# B&R Automation Studio project TD52 (part 59)

#### AC_SS.c
```c
/********************************************************************
 * COPYRIGHT -- Bernecker + Rainer Industrie-Elektronik Ges.m.b.H.
 ********************************************************************
 * Program: AC_SS
 * File: AC_SS.c
 * Author: 105055527
 * Created: Thu May 19 13:50:06 2016
 ********************************************************************
 * Implementation of program AC_SS
 ********************************************************************
 * Generated with B&R Automation Studio Target for Simulink V5.0
 * (ERT based)
 ********************************************************************/
#include "AC_SS.h"
#include "AC_SS_private.h"

/*  Defines */

/*  Data Types */

/**************************** GLOBAL DATA *************************************/
/*  Definitions */

/*  Declarations  */

/***************************** FILE SCOPE DATA ********************************/

/*************************** FUNCTIONS ****************************************/

/*
 * Initial conditions for atomic system:
 *    '<S13>/Filter'
 *    '<S19>/Filter'
 *    '<S25>/Filter'
 *    '<S31>/Filter'
 *    '<S37>/Filter'
 *    '<S43>/Filter'
 *    '<S49>/Filter'
 *    '<S55>/Filter'
 */
void AC_SS_Filter_Init(real32_T rtu_x0, rtDW_Filter_AC_SS *localDW, struct SS* inst)
{
  /* InitializeConditions for DiscreteIntegrator: '<S14>/Discrete-Time Integrator' */
  localDW->DiscreteTimeIntegrator_DSTATE = rtu_x0;
}

/*
 * Output and update for atomic system:
 *    '<S13>/Filter'
 *    '<S19>/Filter'
 *    '<S25>/Filter'
 *    '<S31>/Filter'
 *    '<S37>/Filter'
 *    '<S43>/Filter'
 *    '<S49>/Filter'
 *    '<S55>/Filter'
 */
void AC_SS_Filter(real32_T rtu_in, real32_T rtu_T_filt, boolean_T rtu_reset,
                  real32_T rtu_x0, rtB_Filter_AC_SS *localB, rtDW_Filter_AC_SS
                  *localDW, struct SS* inst)
{
  /* local block i/o variables */
  real32_T rtb_Divide4;
  real32_T tmp;

  /* Switch: '<S15>/Switch' incorporates:
   *  Abs: '<S15>/Abs'
   *  RelationalOperator: '<S15>/Relational Operator'
   */
  if (2.22044605E-16F >= (real32_T)fabs(rtu_T_filt)) {
    tmp = 2.22044605E-16F;
  } else {
    tmp = rtu_T_filt;
  }

  /* End of Switch: '<S15>/Switch' */

  /* Product: '<S14>/Divide4' incorporates:
   *  Sum: '<S14>/Sum4'
   */
  rtb_Divide4 = (rtu_in - localDW->DiscreteTimeIntegrator_DSTATE) / tmp;

  /* DiscreteIntegrator: '<S14>/Discrete-Time Integrator' */
  if (rtu_reset || (localDW->DiscreteTimeIntegrator_PrevRese != 0)) {
    localDW->DiscreteTimeIntegrator_DSTATE = rtu_x0;
  }

  localB->DiscreteTimeIntegrator = 0.005F * rtb_Divide4 +
    localDW->DiscreteTimeIntegrator_DSTATE;

  /* End of DiscreteIntegrator: '<S14>/Discrete-Time Integrator' */

  /* Update for DiscreteIntegrator: '<S14>/Discrete-Time Integrator' */
  if (!rtu_reset) {
    localDW->DiscreteTimeIntegrator_DSTATE = 0.005F * rtb_Divide4 +
      localB->DiscreteTimeIntegrator;
  }

  if (rtu_reset) {
    localDW->DiscreteTimeIntegrator_PrevRese = 1;
  } else {
    localDW->DiscreteTimeIntegrator_PrevRese = 0;
  }

  /* End of Update for DiscreteIntegrator: '<S14>/Discrete-Time Integrator' */
}

/* Model step function */
void AC_SS_step(struct BlockIO_AC_SS *AC_SS_B, struct D_Work_AC_SS *AC_SS_DWork,
                ExternalOutputs_AC_SS *AC_SS_Y, struct SS* inst)
{
  /* local block i/o variables */
  real32_T rtb_rAct;
  real32_T rtb_rTi_Filt;
  real32_T rtb_rAct_h;
  real32_T rtb_rTi_Filt_h;
  real32_T rtb_rAct_hj;
  real32_T rtb_rTi_Filt_l;
  real32_T rtb_rAct_g;
  real32_T rtb_rTi_Filt_j;
  real32_T rtb_rAct_n;
  real32_T rtb_rTi_Filt_e;
  real32_T rtb_rAct_b;
  real32_T rtb_rTi_Filt_i;
  real32_T rtb_rAct_d;
  real32_T rtb_rTi_Filt_k;
  real32_T rtb_rAct_i;
  real32_T rtb_rTi_Filt_m;
  boolean_T rtb_bReset;
  real32_T rtb_Abs;
  boolean_T rtb_RelationalOperator5;
  boolean_T rtb_RelationalOperator1;
  boolean_T rtb_RelationalOperator5_n;
  boolean_T rtb_RelationalOperator1_m;
  boolean_T rtb_RelationalOperator5_p;
  boolean_T rtb_RelationalOperator1_a;
  boolean_T rtb_RelationalOperator5_b;
  boolean_T rtb_RelationalOperator1_d;
  boolean_T rtb_RelationalOperator5_j;
  boolean_T rtb_RelationalOperator1_am;
  boolean_T rtb_RelationalOperator5_j2;
  boolean_T rtb_RelationalOperator1_p;
  boolean_T rtb_RelationalOperator5_e;
  boolean_T rtb_RelationalOperator1_n;
  boolean_T rtb_RelationalOperator5_m;
  boolean_T tmp[8];
  uint8_T tmp_0;
  int32_T i;
  boolean_T tmp_1[8];

  /* S-Function (bur_bus_in): '<Root>/Bus Input' */
  AC_SS_B->BusInput = inst->in;

  /* BusSelector: '<S2>/Bus Selector2' */
  rtb_bReset = AC_SS_B->BusInput.bReset;

  /* BusSelector: '<S7>/Bus Selector' */
  rtb_rAct = AC_SS_B->BusInput.P2s.rAct;
  rtb_rTi_Filt = AC_SS_B->BusInput.P2s.rTi_Filt;

  /* Sum: '<S36>/Add3' */
  rtb_Abs = AC_SS_B->BusInput.P2s.rSet - rtb_rAct;

  /* Abs: '<S36>/Abs3' */
  rtb_Abs = (real32_T)fabs(rtb_Abs);

  /* RelationalOperator: '<S36>/Relational Operator5' */
  rtb_RelationalOperator5 = (rtb_Abs <= AC_SS_B->BusInput.P2s.rAbsLim);

  /* Outputs for Atomic SubSystem: '<S37>/Filter' */
  AC_SS_Filter(rtb_rAct, rtb_rTi_Filt, rtb_bReset, AC_SS_ConstB.Constant,
               &AC_SS_B->Filter, &AC_SS_DWork->Filter, inst);

  /* End of Outputs for SubSystem: '<S37>/Filter' */

  /* Sum: '<S37>/Add' */
  rtb_Abs = rtb_rAct - AC_SS_B->Filter.DiscreteTimeIntegrator;

  /* Abs: '<S37>/Abs' */
  rtb_Abs = (real32_T)fabs(rtb_Abs);

  /* RelationalOperator: '<S37>/Relational Operator1' */
  rtb_RelationalOperator1 = (rtb_Abs <= AC_SS_B->BusInput.P2s.rRelLim);

  /* BusSelector: '<S9>/Bus Selector' */
  rtb_rAct_h = AC_SS_B->BusInput.T2s.rAct;
  rtb_rTi_Filt_h = AC_SS_B->BusInput.T2s.rTi_Filt;

  /* Sum: '<S48>/Add3' */
  rtb_Abs = AC_SS_B->BusInput.T2s.rSet - rtb_rAct_h;

  /* Abs: '<S48>/Abs3' */
  rtb_Abs = (real32_T)fabs(rtb_Abs);

  /* RelationalOperator: '<S48>/Relational Operator5' */
  rtb_RelationalOperator5_n = (rtb_Abs <= AC_SS_B->BusInput.T2s.rAbsLim);

  /* Outputs for Atomic SubSystem: '<S49>/Filter' */
  AC_SS_Filter(rtb_rAct_h, rtb_rTi_Filt_h, rtb_bReset, AC_SS_ConstB.Constant_d,
               &AC_SS_B->Filter_n, &AC_SS_DWork->Filter_n, inst);

  /* End of Outputs for SubSystem: '<S49>/Filter' */

  /* Sum: '<S49>/Add' */
  rtb_Abs = rtb_rAct_h - AC_SS_B->Filter_n.DiscreteTimeIntegrator;

  /* Abs: '<S49>/Abs' */
  rtb_Abs = (real32_T)fabs(rtb_Abs);

  /* RelationalOperator: '<S49>/Relational Operator1' */
  rtb_RelationalOperator1_m = (rtb_Abs <= AC_SS_B->BusInput.T2s.rRelLim);

  /* BusSelector: '<S10>/Bus Selector' */
  rtb_rAct_hj = AC_SS_B->BusInput.T_EG.rAct;
  rtb_rTi_Filt_l = AC_SS_B->BusInput.T_EG.rTi_Filt;

  /* Sum: '<S54>/Add3' */
  rtb_Abs = AC_SS_B->BusInput.T_EG.rSet - rtb_rAct_hj;

  /* Abs: '<S54>/Abs3' */
  rtb_Abs = (real32_T)fabs(rtb_Abs);

  /* RelationalOperator: '<S54>/Relational Operator5' */
  rtb_RelationalOperator5_p = (rtb_Abs <= AC_SS_B->BusInput.T_EG.rAbsLim);

  /* Outputs for Atomic SubSystem: '<S55>/Filter' */
  AC_SS_Filter(rtb_rAct_hj, rtb_rTi_Filt_l, rtb_bReset, AC_SS_ConstB.Constant_j,
               &AC_SS_B->Filter_c, &AC_SS_DWork->Filter_c, inst);

  /* End of Outputs for SubSystem: '<S55>/Filter' */

  /* Sum: '<S55>/Add' */
  rtb_Abs = rtb_rAct_hj - AC_SS_B->Filter_c.DiscreteTimeIntegrator;

  /* Abs: '<S55>/Abs' */
  rtb_Abs = (real32_T)fabs(rtb_Abs);

  /* RelationalOperator: '<S55>/Relational Operator1' */
  rtb_RelationalOperator1_a = (rtb_Abs <= AC_SS_B->BusInput.T_EG.rRelLim);

  /* BusSelector: '<S6>/Bus Selector' */
  rtb_rAct_g = AC_SS_B->BusInput.P_Norm.rAct;
  rtb_rTi_Filt_j = AC_SS_B->BusInput.P_Norm.rTi_Filt;

  /* Sum: '<S30>/Add3' */
  rtb_Abs = AC_SS_B->BusInput.P_Norm.rSet - rtb_rAct_g;

  /* Abs: '<S30>/Abs3' */
  rtb_Abs = (real32_T)fabs(rtb_Abs);

  /* RelationalOperator: '<S30>/Relational Operator5' */
  rtb_RelationalOperator5_b = (rtb_Abs <= AC_SS_B->BusInput.P_Norm.rAbsLim);

  /* Outputs for Atomic SubSystem: '<S31>/Filter' */
  AC_SS_Filter(rtb_rAct_g, rtb_rTi_Filt_j, rtb_bReset, AC_SS_ConstB.Constant_h,
               &AC_SS_B->Filter_h, &AC_SS_DWork->Filter_h, inst);

  /* End of Outputs for SubSystem: '<S31>/Filter' */

  /* Sum: '<S31>/Add' */
  rtb_Abs = rtb_rAct_g - AC_SS_B->Filter_h.DiscreteTimeIntegrator;

  /* Abs: '<S31>/Abs' */
  rtb_Abs = (real32_T)fabs(rtb_Abs);

  /* RelationalOperator: '<S31>/Relational Operator1' */
  rtb_RelationalOperator1_d = (rtb_Abs <= AC_SS_B->BusInput.P_Norm.rRelLim);

  /* BusSelector: '<S4>/Bus Selector' */
  rtb_rAct_n = AC_SS_B->BusInput.Lam.rAct;
  rtb_rTi_Filt_e = AC_SS_B->BusInput.Lam.rTi_Filt;

  /* Sum: '<S18>/Add3' */
  rtb_Abs = AC_SS_B->BusInput.Lam.rSet - rtb_rAct_n;

  /* Abs: '<S18>/Abs3' */
  rtb_Abs = (real32_T)fabs(rtb_Abs);

  /* RelationalOperator: '<S18>/Relational Operator5' */
  rtb_RelationalOperator5_j = (rtb_Abs <= AC_SS_B->BusInput.Lam.rAbsLim);

  /* Outputs for Atomic SubSystem: '<S19>/Filter' */
  AC_SS_Filter(rtb_rAct_n, rtb_rTi_Filt_e, rtb_bReset, AC_SS_ConstB.Constant_g,
               &AC_SS_B->Filter_a, &AC_SS_DWork->Filter_a, inst);

  /* End of Outputs for SubSystem: '<S19>/Filter' */

  /* Sum: '<S19>/Add' */
  rtb_Abs = rtb_rAct_n - AC_SS_B->Filter_a.DiscreteTimeIntegrator;

  /* Abs: '<S19>/Abs' */
  rtb_Abs = (real32_T)fabs(rtb_Abs);

  /* RelationalOperator: '<S19>/Relational Operator1' */
  rtb_RelationalOperator1_am = (rtb_Abs <= AC_SS_B->BusInput.Lam.rRelLim);

  /* BusSelector: '<S5>/Bus Selector' */
  rtb_rAct_b = AC_SS_B->BusInput.N_Norm.rAct;
  rtb_rTi_Filt_i = AC_SS_B->BusInput.N_Norm.rTi_Filt;

  /* Sum: '<S24>/Add3' */
  rtb_Abs = AC_SS_B->BusInput.N_Norm.rSet - rtb_rAct_b;

  /* Abs: '<S24>/Abs3' */
  rtb_Abs = (real32_T)fabs(rtb_Abs);

  /* RelationalOperator: '<S24>/Relational Operator5' */
  rtb_RelationalOperator5_j2 = (rtb_Abs <= AC_SS_B->BusInput.N_Norm.rAbsLim);

  /* Outputs for Atomic SubSystem: '<S25>/Filter' */
  AC_SS_Filter(rtb_rAct_b, rtb_rTi_Filt_i, rtb_bReset, AC_SS_ConstB.Constant_hq,
               &AC_SS_B->Filter_e, &AC_SS_DWork->Filter_e, inst);

  /* End of Outputs for SubSystem: '<S25>/Filter' */

  /* Sum: '<S25>/Add' */
  rtb_Abs = rtb_rAct_b - AC_SS_B->Filter_e.DiscreteTimeIntegrator;

  /* Abs: '<S25>/Abs' */
  rtb_Abs = (real32_T)fabs(rtb_Abs);

  /* RelationalOperator: '<S25>/Relational Operator1' */
  rtb_RelationalOperator1_p = (rtb_Abs <= AC_SS_B->BusInput.N_Norm.rRelLim);

  /* BusSelector: '<S8>/Bus Selector' */
  rtb_rAct_d = AC_SS_B->BusInput.P_d_Norm.rAct;
  rtb_rTi_Filt_k = AC_SS_B->BusInput.P_d_Norm.rTi_Filt;

  /* Sum: '<S42>/Add3' */
  rtb_Abs = AC_SS_B->BusInput.P_d_Norm.rSet - rtb_rAct_d;

  /* Abs: '<S42>/Abs3' */
  rtb_Abs = (real32_T)fabs(rtb_Abs);

  /* RelationalOperator: '<S42>/Relational Operator5' */
  rtb_RelationalOperator5_e = (rtb_Abs <= AC_SS_B->BusInput.P_d_Norm.rAbsLim);

  /* Outputs for Atomic SubSystem: '<S43>/Filter' */
  AC_SS_Filter(rtb_rAct_d, rtb_rTi_Filt_k, rtb_bReset, AC_SS_ConstB.Constant_b,
               &AC_SS_B->Filter_f, &AC_SS_DWork->Filter_f, inst);

  /* End of Outputs for SubSystem: '<S43>/Filter' */

  /* Sum: '<S43>/Add' */
  rtb_Abs = rtb_rAct_d - AC_SS_B->Filter_f.DiscreteTimeIntegrator;

  /* Abs: '<S43>/Abs' */
  rtb_Abs = (real32_T)fabs(rtb_Abs);

  /* RelationalOperator: '<S43>/Relational Operator1' */
  rtb_RelationalOperator1_n = (rtb_Abs <= AC_SS_B->BusInput.P_d_Norm.rRelLim);

  /* BusSelector: '<S3>/Bus Selector' */
  rtb_rAct_i = AC_SS_B->BusInput.IP.rAct;
  rtb_rTi_Filt_m = AC_SS_B->BusInput.IP.rTi_Filt;

  /* Sum: '<S12>/Add3' */
  rtb_Abs = AC_SS_B->BusInput.IP.rSet - rtb_rAct_i;

  /* Abs: '<S12>/Abs3' */
  rtb_Abs = (real32_T)fabs(rtb_Abs);

  /* RelationalOperator: '<S12>/Relational Operator5' */
  rtb_RelationalOperator5_m = (rtb_Abs <= AC_SS_B->BusInput.IP.rAbsLim);

  /* Outputs for Atomic SubSystem: '<S13>/Filter' */
  AC_SS_Filter(rtb_rAct_i, rtb_rTi_Filt_m, rtb_bReset, AC_SS_ConstB.Constant_f,
               &AC_SS_B->Filter_o, &AC_SS_DWork->Filter_o, inst);

  /* End of Outputs for SubSystem: '<S13>/Filter' */

  /* Sum: '<S13>/Add' */
  rtb_Abs = rtb_rAct_i - AC_SS_B->Filter_o.DiscreteTimeIntegrator;

  /* Abs: '<S13>/Abs' */
  rtb_Abs = (real32_T)fabs(rtb_Abs);

  /* BusCreator: '<S2>/Bus Creator1' incorporates:
   *  BusCreator: '<S10>/Bus Creator2'
   *  BusCreator: '<S3>/Bus Creator2'
   *  BusCreator: '<S4>/Bus Creator2'
   *  BusCreator: '<S5>/Bus Creator2'
   *  BusCreator: '<S6>/Bus Creator2'
   *  BusCreator: '<S7>/Bus Creator2'
   *  BusCreator: '<S8>/Bus Creator2'
   *  BusCreator: '<S9>/Bus Creator2'
   *  RelationalOperator: '<S13>/Relational Operator1'
   */
  AC_SS_Y->dbg.P2s.bAbs = rtb_RelationalOperator5;
  AC_SS_Y->dbg.P2s.bRel = rtb_RelationalOperator1;
  AC_SS_Y->dbg.T2s.bAbs = rtb_RelationalOperator5_n;
  AC_SS_Y->dbg.T2s.bRel = rtb_RelationalOperator1_m;
  AC_SS_Y->dbg.T_EG.bAbs = rtb_RelationalOperator5_p;
  AC_SS_Y->dbg.T_EG.bRel = rtb_RelationalOperator1_a;
  AC_SS_Y->dbg.P_Norm.bAbs = rtb_RelationalOperator5_b;
  AC_SS_Y->dbg.P_Norm.bRel = rtb_RelationalOperator1_d;
  AC_SS_Y->dbg.Lam.bAbs = rtb_RelationalOperator5_j;
  AC_SS_Y->dbg.Lam.bRel = rtb_RelationalOperator1_am;
  AC_SS_Y->dbg.N_Norm.bAbs = rtb_RelationalOperator5_j2;
  AC_SS_Y->dbg.N_Norm.bRel = rtb_RelationalOperator1_p;
  AC_SS_Y->dbg.P_d_Norm.bAbs = rtb_RelationalOperator5_e;
  AC_SS_Y->dbg.P_d_Norm.bRel = rtb_RelationalOperator1_n;
  AC_SS_Y->dbg.IP.bAbs = rtb_RelationalOperator5_m;
  AC_SS_Y->dbg.IP.bRel = (rtb_Abs <= AC_SS_B->BusInput.IP.rRelLim);

  /* SignalConversion: '<S2>/TmpSignal ConversionAtGainInport1' incorporates:
   *  BusSelector: '<S2>/Bus Selector'
   */
  tmp[0] = AC_SS_Y->dbg.P2s.bAbs;
  tmp[1] = AC_SS_Y->dbg.T2s.bAbs;
  tmp[2] = AC_SS_Y->dbg.T_EG.bAbs;
  tmp[3] = AC_SS_Y->dbg.P_Norm.bAbs;
  tmp[4] = AC_SS_Y->dbg.Lam.bAbs;
  tmp[5] = AC_SS_Y->dbg.N_Norm.bAbs;
  tmp[6] = AC_SS_Y->dbg.P_d_Norm.bAbs;
  tmp[7] = AC_SS_Y->dbg.IP.bAbs;

  /* Gain: '<S2>/Gain' */
  tmp_0 = 0U;
  for (i = 0; i < 8; i++) {
    tmp_0 = (uint8_T)((uint32_T)tmp_0 + (uint32_T)(tmp[i] ?
      AC_SS_ConstP.pooled4[i] : 0));
  }

  /* Outport: '<Root>/iAbs' incorporates:
   *  Gain: '<S2>/Gain'
   */
  AC_SS_Y->iAbs = tmp_0;

  /* SignalConversion: '<S2>/TmpSignal ConversionAtGain1Inport1' incorporates:
   *  BusSelector: '<S2>/Bus Selector1'
   */
  tmp_1[0] = AC_SS_Y->dbg.P2s.bRel;
  tmp_1[1] = AC_SS_Y->dbg.T2s.bRel;
  tmp_1[2] = AC_SS_Y->dbg.T_EG.bRel;
  tmp_1[3] = AC_SS_Y->dbg.P_Norm.bRel;
  tmp_1[4] = AC_SS_Y->dbg.Lam.bRel;
  tmp_1[5] = AC_SS_Y->dbg.N_Norm.bRel;
  tmp_1[6] = AC_SS_Y->dbg.P_d_Norm.bRel;
  tmp_1[7] = AC_SS_Y->dbg.IP.bRel;

  /* Gain: '<S2>/Gain1' */
  tmp_0 = 0U;
  for (i = 0; i < 8; i++) {
    tmp_0 = (uint8_T)((uint32_T)tmp_0 + (uint32_T)(tmp_1[i] ?
      AC_SS_ConstP.pooled4[i] : 0));
  }

  /* Outport: '<Root>/iRel' incorporates:
   *  Gain: '<S2>/Gain1'
   */
  AC_SS_Y->iRel = tmp_0;

  /* S-Function (bur_bus_out): '<Root>/Bus Output' */
  inst->dbg = AC_SS_Y->dbg;

  /* S-Function (bur_out): '<Root>/Output' */
  inst->iAbs = AC_SS_Y->iAbs;

  /* S-Function (bur_out): '<Root>/Output1' */
  inst->iRel = AC_SS_Y->iRel;
}

/* Model initialize function */
void AC_SS_initialize(struct D_Work_AC_SS *AC_SS_DWork, struct SS* inst)
{
  /* InitializeConditions for Atomic SubSystem: '<S37>/Filter' */
  AC_SS_Filter_Init(AC_SS_ConstB.Constant, &AC_SS_DWork->Filter, inst);

  /* End of InitializeConditions for SubSystem: '<S37>/Filter' */

  /* InitializeConditions for Atomic SubSystem: '<S49>/Filter' */
  AC_SS_Filter_Init(AC_SS_ConstB.Constant_d, &AC_SS_DWork->Filter_n, inst);

  /* End of InitializeConditions for SubSystem: '<S49>/Filter' */

  /* InitializeConditions for Atomic SubSystem: '<S55>/Filter' */
  AC_SS_Filter_Init(AC_SS_ConstB.Constant_j, &AC_SS_DWork->Filter_c, inst);

  /* End of InitializeConditions for SubSystem: '<S55>/Filter' */

  /* InitializeConditions for Atomic SubSystem: '<S31>/Filter' */
  AC_SS_Filter_Init(AC_SS_ConstB.Constant_h, &AC_SS_DWork->Filter_h, inst);

  /* End of InitializeConditions for SubSystem: '<S31>/Filter' */

  /* InitializeConditions for Atomic SubSystem: '<S19>/Filter' */
  AC_SS_Filter_Init(AC_SS_ConstB.Constant_g, &AC_SS_DWork->Filter_a, inst);

  /* End of InitializeConditions for SubSystem: '<S19>/Filter' */

  /* InitializeConditions for Atomic SubSystem: '<S25>/Filter' */
  AC_SS_Filter_Init(AC_SS_ConstB.Constant_hq, &AC_SS_DWork->Filter_e, inst);

  /* End of InitializeConditions for SubSystem: '<S25>/Filter' */

  /* InitializeConditions for Atomic SubSystem: '<S43>/Filter' */
  AC_SS_Filter_Init(AC_SS_ConstB.Constant_b, &AC_SS_DWork->Filter_f, inst);

  /* End of InitializeConditions for SubSystem: '<S43>/Filter' */

  /* InitializeConditions for Atomic SubSystem: '<S13>/Filter' */
  AC_SS_Filter_Init(AC_SS_ConstB.Constant_f, &AC_SS_DWork->Filter_o, inst);

  /* End of InitializeConditions for SubSystem: '<S13>/Filter' */
}

/* Model terminate function */
void AC_SS_terminate(struct SS* inst)
{
  /* (no terminate code required) */
}

/*======================== TOOL VERSION INFORMATION ==========================*
 * MATLAB 8.0 (R2012b)20-Jul-2012                                             *
 * Simulink 8.0 (R2012b)20-Jul-2012                                           *
 * Simulink Coder 8.3 (R2012b)20-Jul-2012                                     *
 * Embedded Coder 6.3 (R2012b)20-Jul-2012                                     *
 * Stateflow 8.0 (R2012b)20-Jul-2012                                          *
 *============================================================================*/

/*======================= LICENSE IN USE INFORMATION =========================*
 * matlab                                                                     *
 * matlab_coder                                                               *
 * real-time_workshop                                                         *
 * rtw_embedded_coder                                                         *
 * simulink                                                                   *
 *============================================================================*/
```

#### AC_SS.h
```c
/********************************************************************
 * COPYRIGHT -- Bernecker + Rainer Industrie-Elektronik Ges.m.b.H.
 ********************************************************************
 * Program: AC_SS
 * File: AC_SS.h
 * Author: 105055527
 * Created: Thu May 19 13:50:06 2016
 ********************************************************************
 * Header for program AC_SS
 ********************************************************************
 * Generated with B&R Automation Studio Target for Simulink V5.0
 * (ERT based)
 ********************************************************************/

#ifndef RTW_HEADER_AC_SS_h_
#define RTW_HEADER_AC_SS_h_
#ifndef AC_SS_COMMON_INCLUDES_
# define AC_SS_COMMON_INCLUDES_
#include <math.h>
#include "rtwtypes.h"
#endif                                 /* AC_SS_COMMON_INCLUDES_ */

#include "AC_SS_types.h"
#include "lSS.h"

/* Macros for accessing real-time model data structure */
#ifndef rtmGetErrorStatus
# define rtmGetErrorStatus(rtm)        ((rtm)->errorStatus)
#endif

#ifndef rtmSetErrorStatus
# define rtmSetErrorStatus(rtm, val)   ((rtm)->errorStatus = (val))
#endif

#ifndef rtmGetStopRequested
# define rtmGetStopRequested(rtm)      ((void*) 0)
#endif

#ifndef MIN
#define MIN(a,b)                       ((a) < (b) ? (a) : (b))
#endif

#ifndef MAX
#define MAX(a,b)                       ((a) > (b) ? (a) : (b))
#endif

/* Block signals for system '<S13>/Filter' */

/* Block states (auto storage) for system '<S13>/Filter' */

/* Block signals (auto storage) */

/* Block states (auto storage) for system '<Root>' */

/* Invariant block signals for system '<S13>/Filter' */

/* Invariant block signals (auto storage) */

/* Constant parameters (auto storage) */

/* External outputs (root outports fed by signals with auto storage) */

/* Real-time Model Data Structure */

extern const ConstBlockIO_AC_SS AC_SS_ConstB;/* constant block i/o */

/* Constant parameters (auto storage) */
extern const ConstParam_AC_SS AC_SS_ConstP;

/* Model entry point functions */
extern void AC_SS_initialize(D_Work_AC_SS *AC_SS_DWork, struct SS* inst);
extern void AC_SS_step(BlockIO_AC_SS *AC_SS_B, D_Work_AC_SS *AC_SS_DWork,
  ExternalOutputs_AC_SS *AC_SS_Y, struct SS* inst);
extern void AC_SS_terminate(struct SS* inst);

/*-
 * The generated code includes comments that allow you to trace directly
 * back to the appropriate location in the model.  The basic format
 * is <system>/block_name, where system is the system number (uniquely
 * assigned by Simulink) and block_name is the name of the block.
 *
 * Use the MATLAB hilite_system command to trace the generated code back
 * to the model.  For example,
 *
 * hilite_system('<S3>')    - opens system 3
 * hilite_system('<S3>/Kp') - opens and selects block Kp which resides in S3
 *
 * Here is the system hierarchy for this model
 *
 * '<Root>' : 'AC_SS'
 * '<S1>'   : 'AC_SS/Environment Controller'
 * '<S2>'   : 'AC_SS/SS'
 * '<S3>'   : 'AC_SS/SS/SS_IP'
 * '<S4>'   : 'AC_SS/SS/SS_Lam'
 * '<S5>'   : 'AC_SS/SS/SS_N'
 * '<S6>'   : 'AC_SS/SS/SS_P'
 * '<S7>'   : 'AC_SS/SS/SS_P2s'
 * '<S8>'   : 'AC_SS/SS/SS_P_d'
 * '<S9>'   : 'AC_SS/SS/SS_T2s'
 * '<S10>'  : 'AC_SS/SS/SS_T_EG'
 * '<S11>'  : 'AC_SS/SS/SS_IP/SS'
 * '<S12>'  : 'AC_SS/SS/SS_IP/SS/Deviation_comp1'
 * '<S13>'  : 'AC_SS/SS/SS_IP/SS/Slew_rate_comp3'
 * '<S14>'  : 'AC_SS/SS/SS_IP/SS/Slew_rate_comp3/Filter'
 * '<S15>'  : 'AC_SS/SS/SS_IP/SS/Slew_rate_comp3/Filter/Divisor'
 * '<S16>'  : 'AC_SS/SS/SS_IP/SS/Slew_rate_comp3/Filter/Divisor/Data Type Conversion Inherited'
 * '<S17>'  : 'AC_SS/SS/SS_Lam/SS'
 * '<S18>'  : 'AC_SS/SS/SS_Lam/SS/Deviation_comp1'
 * '<S19>'  : 'AC_SS/SS/SS_Lam/SS/Slew_rate_comp3'
 * '<S20>'  : 'AC_SS/SS/SS_Lam/SS/Slew_rate_comp3/Filter'
 * '<S21>'  : 'AC_SS/SS/SS_Lam/SS/Slew_rate_comp3/Filter/Divisor'
 * '<S22>'  : 'AC_SS/SS/SS_Lam/SS/Slew_rate_comp3/Filter/Divisor/Data Type Conversion Inherited'
 * '<S23>'  : 'AC_SS/SS/SS_N/SS'
 * '<S24>'  : 'AC_SS/SS/SS_N/SS/Deviation_comp1'
 * '<S25>'  : 'AC_SS/SS/SS_N/SS/Slew_rate_comp3'
 * '<S26>'  : 'AC_SS/SS/SS_N/SS/Slew_rate_comp3/Filter'
 * '<S27>'  : 'AC_SS/SS/SS_N/SS/Slew_rate_comp3/Filter/Divisor'
 * '<S28>'  : 'AC_SS/SS/SS_N/SS/Slew_rate_comp3/Filter/Divisor/Data Type Conversion Inherited'
 * '<S29>'  : 'AC_SS/SS/SS_P/SS'
 * '<S30>'  : 'AC_SS/SS/SS_P/SS/Deviation_comp1'
 * '<S31>'  : 'AC_SS/SS/SS_P/SS/Slew_rate_comp3'
 * '<S32>'  : 'AC_SS/SS/SS_P/SS/Slew_rate_comp3/Filter'
 * '<S33>'  : 'AC_SS/SS/SS_P/SS/Slew_rate_comp3/Filter/Divisor'
 * '<S34>'  : 'AC_SS/SS/SS_P/SS/Slew_rate_comp3/Filter/Divisor/Data Type Conversion Inherited'
 * '<S35>'  : 'AC_SS/SS/SS_P2s/SS'
 * '<S36>'  : 'AC_SS/SS/SS_P2s/SS/Deviation_comp1'
 * '<S37>'  : 'AC_SS/SS/SS_P2s/SS/Slew_rate_comp3'
 * '<S38>'  : 'AC_SS/SS/SS_P2s/SS/Slew_rate_comp3/Filter'
 * '<S39>'  : 'AC_SS/SS/SS_P2s/SS/Slew_rate_comp3/Filter/Divisor'
 * '<S40>'  : 'AC_SS/SS/SS_P2s/SS/Slew_rate_comp3/Filter/Divisor/Data Type Conversion Inherited'
 * '<S41>'  : 'AC_SS/SS/SS_P_d/SS'
 * '<S42>'  : 'AC_SS/SS/SS_P_d/SS/Deviation_comp1'
 * '<S43>'  : 'AC_SS/SS/SS_P_d/SS/Slew_rate_comp3'
 * '<S44>'  : 'AC_SS/SS/SS_P_d/SS/Slew_rate_comp3/Filter'
 * '<S45>'  : 'AC_SS/SS/SS_P_d/SS/Slew_rate_comp3/Filter/Divisor'
 * '<S46>'  : 'AC_SS/SS/SS_P_d/SS/Slew_rate_comp3/Filter/Divisor/Data Type Conversion Inherited'
 * '<S47>'  : 'AC_SS/SS/SS_T2s/SS'
 * '<S48>'  : 'AC_SS/SS/SS_T2s/SS/Deviation_comp1'
 * '<S49>'  : 'AC_SS/SS/SS_T2s/SS/Slew_rate_comp3'
 * '<S50>'  : 'AC_SS/SS/SS_T2s/SS/Slew_rate_comp3/Filter'
 * '<S51>'  : 'AC_SS/SS/SS_T2s/SS/Slew_rate_comp3/Filter/Divisor'
 * '<S52>'  : 'AC_SS/SS/SS_T2s/SS/Slew_rate_comp3/Filter/Divisor/Data Type Conversion Inherited'
 * '<S53>'  : 'AC_SS/SS/SS_T_EG/SS'
 * '<S54>'  : 'AC_SS/SS/SS_T_EG/SS/Deviation_comp1'
 * '<S55>'  : 'AC_SS/SS/SS_T_EG/SS/Slew_rate_comp3'
 * '<S56>'  : 'AC_SS/SS/SS_T_EG/SS/Slew_rate_comp3/Filter'
 * '<S57>'  : 'AC_SS/SS/SS_T_EG/SS/Slew_rate_comp3/Filter/Divisor'
 * '<S58>'  : 'AC_SS/SS/SS_T_EG/SS/Slew_rate_comp3/Filter/Divisor/Data Type Conversion Inherited'
 */
#endif                                 /* RTW_HEADER_AC_SS_h_ */
```

#### AC_SS_data.c
```c
/********************************************************************
 * COPYRIGHT -- Bernecker + Rainer Industrie-Elektronik Ges.m.b.H.
 ********************************************************************
 * Program: AC_SS
 * File: AC_SS_data.c
 * Author: 105055527
 * Created: Thu May 19 13:50:06 2016
 ********************************************************************
 * Data for program AC_SS
 ********************************************************************
 * Generated with B&R Automation Studio Target for Simulink V5.0
 * (ERT based)
 ********************************************************************/
#include "AC_SS.h"
#include "AC_SS_private.h"

/*  GLOBAL DATA DEFINITIONS */

/* Invariant block signals (auto storage) */
const ConstBlockIO_AC_SS AC_SS_ConstB = {
  0.0F
  ,                                    /* '<S37>/Constant' */
  0.0F
  ,                                    /* '<S49>/Constant' */
  0.0F
  ,                                    /* '<S55>/Constant' */
  0.0F
  ,                                    /* '<S31>/Constant' */
  0.0F
  ,                                    /* '<S19>/Constant' */
  0.0F
  ,                                    /* '<S25>/Constant' */
  0.0F
  ,                                    /* '<S43>/Constant' */
  0.0F
  ,                                    /* '<S13>/Constant' */

  /* Start of '<S55>/Filter' */
  {
    2.22044605E-16F
    /* '<S58>/Conversion' */
  }
  /* End of '<S55>/Filter' */
  ,

  /* Start of '<S49>/Filter' */
  {
    2.22044605E-16F
    /* '<S52>/Conversion' */
  }
  /* End of '<S49>/Filter' */
  ,

  /* Start of '<S43>/Filter' */
  {
    2.22044605E-16F
    /* '<S46>/Conversion' */
  }
  /* End of '<S43>/Filter' */
  ,

  /* Start of '<S37>/Filter' */
  {
    2.22044605E-16F
    /* '<S40>/Conversion' */
  }
  /* End of '<S37>/Filter' */
  ,

  /* Start of '<S31>/Filter' */
  {
    2.22044605E-16F
    /* '<S34>/Conversion' */
  }
  /* End of '<S31>/Filter' */
  ,

  /* Start of '<S25>/Filter' */
  {
    2.22044605E-16F
    /* '<S28>/Conversion' */
  }
  /* End of '<S25>/Filter' */
  ,

  /* Start of '<S19>/Filter' */
  {
    2.22044605E-16F
    /* '<S22>/Conversion' */
  }
  /* End of '<S19>/Filter' */
  ,

  /* Start of '<S13>/Filter' */
  {
    2.22044605E-16F
    /* '<S16>/Conversion' */
  }
  /* End of '<S13>/Filter' */
};

/* Constant parameters (auto storage) */
const ConstParam_AC_SS AC_SS_ConstP = {
  /* Pooled Parameter (Expression: [1 2 4 8 16 32 64 128])
   * Referenced by:
   *   '<S2>/Gain'
   *   '<S2>/Gain1'
   */
  { 1U, 2U, 4U, 8U, 16U, 32U, 64U, 128U }
};
```

#### AC_SS_private.h
```c
/********************************************************************
 * COPYRIGHT -- Bernecker + Rainer Industrie-Elektronik Ges.m.b.H.
 ********************************************************************
 * Program: AC_SS
 * File: AC_SS_private.h
 * Author: 105055527
 * Created: Thu May 19 13:50:06 2016
 ********************************************************************
 * Header for program AC_SS
 ********************************************************************
 * Generated with B&R Automation Studio Target for Simulink V5.0
 * (ERT based)
 ********************************************************************/

#ifndef RTW_HEADER_AC_SS_private_h_
#define RTW_HEADER_AC_SS_private_h_
#include "rtwtypes.h"
#include <bur/plctypes.h>
#ifndef __RTWTYPES_H__
#error This file requires rtwtypes.h to be included
#else
#ifdef TMWTYPES_PREVIOUSLY_INCLUDED
#error This file requires rtwtypes.h to be included before tmwtypes.h
#else

/* Check for inclusion of an incorrect version of rtwtypes.h */
#ifndef RTWTYPES_ID_C08S16I32L32N32F1
#error This code was generated with a different "rtwtypes.h" than the file included
#endif                                 /* RTWTYPES_ID_C08S16I32L32N32F1 */
#endif                                 /* TMWTYPES_PREVIOUSLY_INCLUDED */
#endif                                 /* __RTWTYPES_H__ */

#ifndef MIN
#define MIN(a,b)                       ((a) < (b) ? (a) : (b))
#endif

#ifndef MAX
#define MAX(a,b)                       ((a) > (b) ? (a) : (b))
#endif

extern void AC_SS_Filter_Init(real32_T rtu_x0, rtDW_Filter_AC_SS *localDW, struct SS* inst);
extern void AC_SS_Filter(real32_T rtu_in, real32_T rtu_T_filt, boolean_T
  rtu_reset, real32_T rtu_x0, rtB_Filter_AC_SS *localB, rtDW_Filter_AC_SS
  *localDW, struct SS* inst);

#endif                                 /* RTW_HEADER_AC_SS_private_h_ */
```

#### AC_SS_types.h
```c
/********************************************************************
 * COPYRIGHT -- Bernecker + Rainer Industrie-Elektronik Ges.m.b.H.
 ********************************************************************
 * Program: AC_SS
 * File: AC_SS_types.h
 * Author: 105055527
 * Created: Thu May 19 13:50:06 2016
 ********************************************************************
 * Header for program AC_SS
 ********************************************************************
 * Generated with B&R Automation Studio Target for Simulink V5.0
 * (ERT based)
 ********************************************************************/

#ifndef RTW_HEADER_AC_SS_types_h_
#define RTW_HEADER_AC_SS_types_h_
#include "rtwtypes.h"
#ifndef MIN
#define MIN(a,b)                       ((a) < (b) ? (a) : (b))
#endif

#ifndef MAX
#define MAX(a,b)                       ((a) > (b) ? (a) : (b))
#endif

/* Forward declaration for rtModel */
typedef struct tag_RTM_AC_SS RT_MODEL_AC_SS;

#endif                                 /* RTW_HEADER_AC_SS_types_h_ */
```

#### SS.c
```c
/********************************************************************
 * COPYRIGHT -- Bernecker + Rainer Industrie-Elektronik Ges.m.b.H.
 ********************************************************************
 * Program: AC_SS
 * File: SS.c
 * Author: 105055527
 * Created: Thu May 19 13:50:06 2016
 ********************************************************************
 * Implementation of program AC_SS
 ********************************************************************
 * Generated with B&R Automation Studio Target for Simulink V5.0
 * (ERT based)
 ********************************************************************/
#include <bur/plctypes.h>
#include "AC_SS.h"
#include "rtwtypes.h"

/* Defines */
#define SS_TERMINATE 4
#define SS_OUTPUT 3
#define SS_INITIALIZE 2

/*  Data Types */

/**************************** GLOBAL DATA *************************************/
/*  Definitions */

/*  Declarations  */

/***************************** FILE SCOPE DATA ********************************/

/*************************** FUNCTIONS ****************************************/
#ifdef __cplusplus

unsigned long bur_heap_size = 6553500;

#endif

void SS(struct SS* inst)
{
/*  tag_RTM_AC_SS* const AC_SS_M = &(inst)->bur_AC_SS;	*/
	BlockIO_AC_SS *AC_SS_B = &(inst)->bur_BlockIO_AC_SS;
	D_Work_AC_SS *AC_SS_DWork = &(inst)->bur_D_Work_AC_SS;
	ExternalOutputs_AC_SS *AC_SS_Y = &(inst)->bur_ExternalOutputs_AC_SS;

  switch (inst->ssMethodType)
  {
   case SS_INITIALIZE:
    /* call model initialize function */
    AC_SS_initialize(AC_SS_DWork, inst);
    break;

   case SS_OUTPUT:
    /* call model step function */
    AC_SS_step(AC_SS_B, AC_SS_DWork, AC_SS_Y, inst);

    break;

   case SS_TERMINATE:
    /* call model terminate function */
    AC_SS_terminate(inst);
    break;
  }
}

/*****************************************************************************
   Function block sample time: 0.01s
 *****************************************************************************/

/*****************************************************************************
   B&R Automation Studio Target for Simulink Version: A5.1.0 (06-May-2016)
 *****************************************************************************/

/*======================== TOOL VERSION INFORMATION ==========================*
 * MATLAB 8.0 (R2012b)20-Jul-2012                                             *
 * Simulink 8.0 (R2012b)20-Jul-2012                                           *
 * Simulink Coder 8.3 (R2012b)20-Jul-2012                                     *
 * Embedded Coder 6.3 (R2012b)20-Jul-2012                                     *
 * Stateflow 8.0 (R2012b)20-Jul-2012                                          *
 *============================================================================*/

/*======================= LICENSE IN USE INFORMATION =========================*
 * matlab                                                                     *
 * matlab_coder                                                               *
 * real-time_workshop                                                         *
 * rtw_embedded_coder                                                         *
 * simulink                                                                   *
 *============================================================================*/
```

### Library Logical/EngineController/Lib_EC/lGen2 (ANSIC, version 1.00.0)

#### Gen2.c
```c
/********************************************************************
 * COPYRIGHT -- B&R Industrial Automation GmbH
 ********************************************************************
 * Program: Gen2_ref
 * File: Gen2.c
 * Author: 105055527
 * Last modified by: kelleto00
 * Created: Wed Apr 16 13:02:53 2008
 * Last modified: Wed Oct 09 10:01:33 2024
 * Model Version: 4.14.00.04
 * Description: V4.10.00.01, 01-09-2020 Keller, Ke Estimator, additive LS factor, Ptraj SpeedCtrl, LVRT Freeze HLCi
   V4.10.00.01, 02-10-2020 Keller, bugfix HLCi p2srefLX init, BDC_lib: change Inf to 1e7
   V4.10.00.01, 13-11-2020 Keller, bugfix LXcorr T2s/ZZP, LSLff damping, dbgOut for Leanox WG compensation
   V4.10.00.01, 27-01-2021 Keller, Lx WGV compensation: no reset in island mode, addition before skipfire compensation
   V4.10.00.01, 02-02-2021 Keller, initialization lambda estimation with rLam_Start
   V4.11.00.01, 28-05-2021 Keller, Gas Quality Change (GQC) Improvements, LHV estimator output
   V4.11.00.01, 05-11-2021 Keller, Bugfix BDC: worksplit offset, optionally Nset instead of Nnom, rN_Eng_LRskipF
   V4.12.00.01, 10-02-2021 Keller, SpeedCtrl2.0 TU Wien: Disturbance Estimator, LQR incl. droop & leanox
   V4.12.00.02, 23-05-2022 Arnold, Leanox point C in low load
   V4.12.00.02, 09-06-2022 Kafka, add external skip fire input for isolated and grid parallel operation
   V4.12.00.03, 15-09-2022 Keller, add power trajectory to HLCi for extended LQR (Droop setpoint)
   V4.12.00.04, 12-10-2022 Keller, add gas flow comp. factor for rejections
   V4.12.00.05, 13-10-2022 Keller, power filter for static skipfire in island mode
   V4.12.00.06, 15-11-2022 Keller, Ke adaptation with disturbance observer
   V4.13.00.01, 15-11-2022 Keller, FDC: R_mix output, HLCi: R_mix for Ke
   V4.13.00.02, 10-07-2023 Keller, interpolation of LHV, rho_gas and Lmin
   V4.13.00.03, 10-07-2023 Keller, load dependent gas dosage delay
   V4.13.00.04, 11-09-2023 Keller, D-part FSM, bugfix dPTV ramp
   V4.13.00.05, 27-02-2024 Keller, Filter outputs without bSS
   V4.13.00.06, 10-04-2024 Keller, bugfix leanox manual mode with bSepEmisCtrl
   V4.14.00.01, 01-07-2024 Keller, iNskip_LRfor Ke calculation
   V4.14.00.02, 17-09-2024 Keller, Use actual speed for observer disturbance dg (Gen2_ref/HLC_Island (HLC_Island_ref)/iLQR_SF/Ref LQR)
   V4.14.00.03, 30-09-2024 Keller, LR gas flow compensation possible without actuator saturation
   V4.14.00.04, 02-10-2024 Keller, Limit derivative power setpoint for FSM
 * modified Comment:
 ********************************************************************
 * Implementation of program Gen2_ref
 ********************************************************************
 * Generated with B&R Automation Studio Target for Simulink V6.7.1
 * (ERT based)
 ********************************************************************/

#include <bur/plctypes.h>
#include "Gen2_ref.h"
#include "rtwtypes.h"

/* Defines */
#define SS_TERMINATE 4
#define SS_OUTPUT 3
#define SS_INITIALIZE 2

/*  Data Types */

/**************************** GLOBAL DATA *************************************/
/*  Definitions */

/*  Declarations  */

/***************************** FILE SCOPE DATA ********************************/

/*************************** FUNCTIONS ****************************************/
#ifdef __cplusplus

unsigned long bur_heap_size = 6553500;

#endif

/*LEGACYMODE_VARIABLES*/
void Gen2(struct Gen2* inst)
{
  tag_RTM_Gen2_ref* const Gen2_ref_M = &(inst)->bur_Gen2_ref;
	inst->bur_Gen2_ref.blockIO = &(inst)->bur_BlockIO_Gen2_ref;
	inst->bur_Gen2_ref.prevZCSigState = &(inst)->bur_PrevZCSigStates_Gen2_ref;
	inst->bur_Gen2_ref.outputs = &(inst)->bur_ExternalOutputs_Gen2_ref;
	inst->bur_Gen2_ref.dwork = &(inst)->bur_D_Work_Gen2_ref;

  switch (inst->ssMethodType)
  {
   case SS_INITIALIZE:
    /* call model initialize function */
    Gen2_ref_initialize(Gen2_ref_M, inst);
    break;

   case SS_OUTPUT:
    /* call model step function */
    Gen2_ref_step(Gen2_ref_M, inst);

    break;

   case SS_TERMINATE:
    /* call model terminate function */
    Gen2_ref_terminate(Gen2_ref_M, inst);
    break;
  }
}

/*****************************************************************************
   Function block sample time: 0.01s
 *****************************************************************************/

/*****************************************************************************
   B&R Automation Studio Target for Simulink Version: A6.7.1 (02-Dec-2022)
 *****************************************************************************/

/*======================== TOOL VERSION INFORMATION ==========================*
 * MATLAB 9.11 (R2021b)14-May-2021                                            *
 * Simulink 10.4 (R2021b)14-May-2021                                          *
 * Simulink Coder 9.6 (R2021b)14-May-2021                                     *
 * Embedded Coder 7.7 (R2021b)14-May-2021                                     *
 * Stateflow 10.5 (R2021b)14-May-2021                                         *
 *============================================================================*/

/*======================= LICENSE IN USE INFORMATION =========================*
 * control_toolbox                                                            *
 * matlab                                                                     *
 * matlab_coder                                                               *
 * real-time_workshop                                                         *
 * rtw_embedded_coder                                                         *
 * simulink                                                                   *
 *============================================================================*/
```
